// SIMATIC S7-200 project (STEP 7-Micro/WIN), CPU 226 CN REL 02.01

ORGANIZATION_BLOCK MAIN:OB1
TITLE=POU Comment
BEGIN
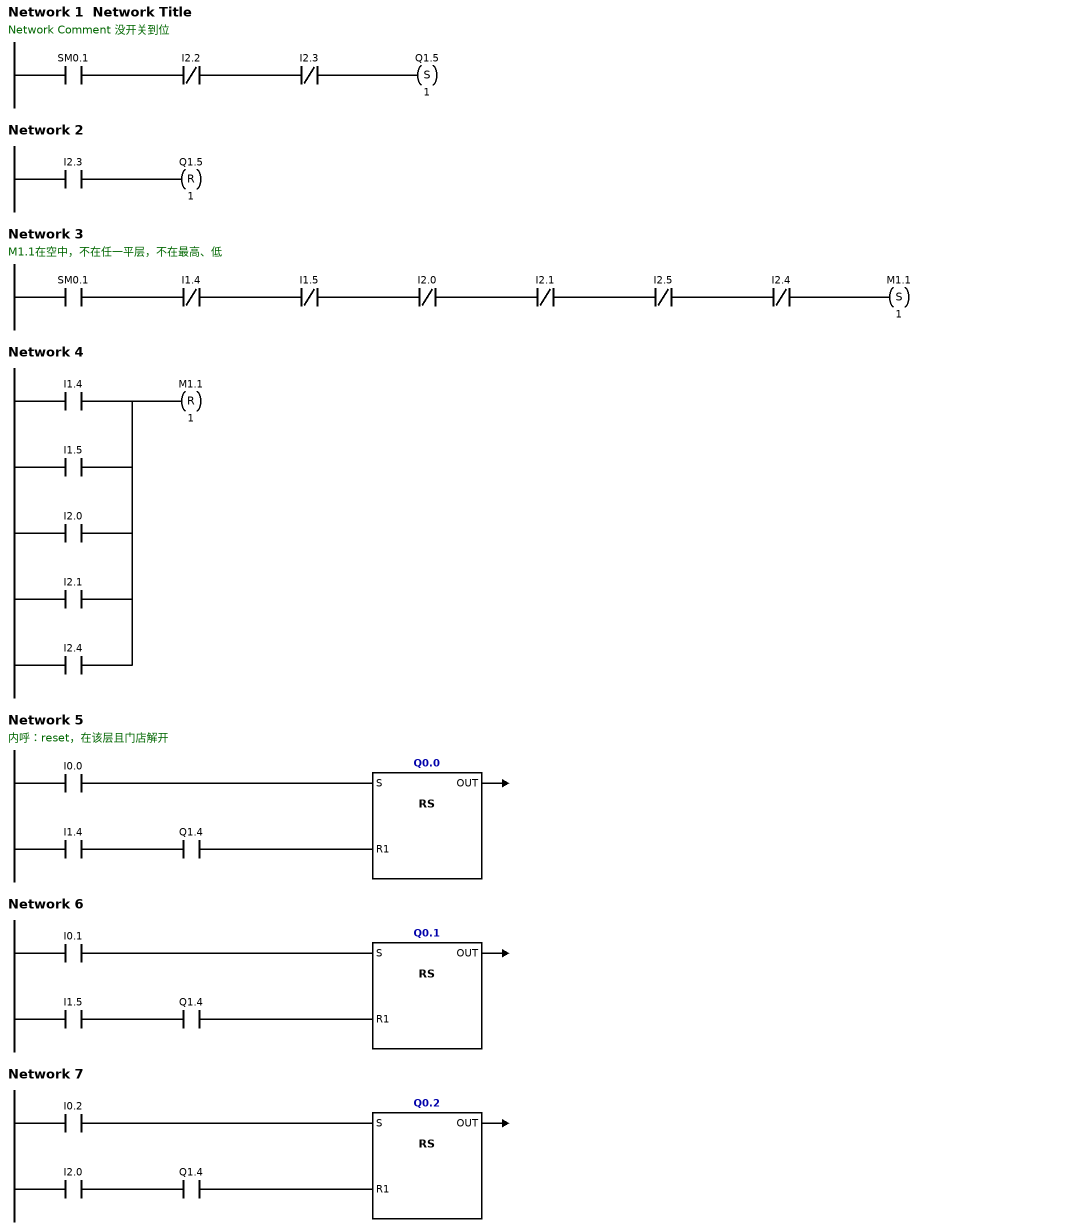
Network 1 // Network Title
// Network Comment 没开关到位
LD     SM0.1
AN     I2.2
AN     I2.3
S      Q1.5, 1
Network 2
LD     I2.3
R      Q1.5, 1
Network 3
// M1.1在空中，不在任一平层，不在最高、低
LD     SM0.1
AN     I1.4
AN     I1.5
AN     I2.0
AN     I2.1
AN     I2.5
AN     I2.4
S      M1.1, 1
Network 4
LD     I1.4
O      I1.5
O      I2.0
O      I2.1
O      I2.4
R      M1.1, 1
Network 5
// 内呼：reset，在该层且门店解开
LD     I0.0
LD     I1.4
A      Q1.4
NOT
LPS
A      Q0.0
=      Q0.0
LPP
ALD
O      Q0.0
=      Q0.0
Network 6
LD     I0.1
LD     I1.5
A      Q1.4
NOT
LPS
A      Q0.1
=      Q0.1
LPP
ALD
O      Q0.1
=      Q0.1
Network 7
LD     I0.2
LD     I2.0
A      Q1.4
NOT
LPS
A      Q0.2
=      Q0.2
LPP
ALD
O      Q0.2
=      Q0.2
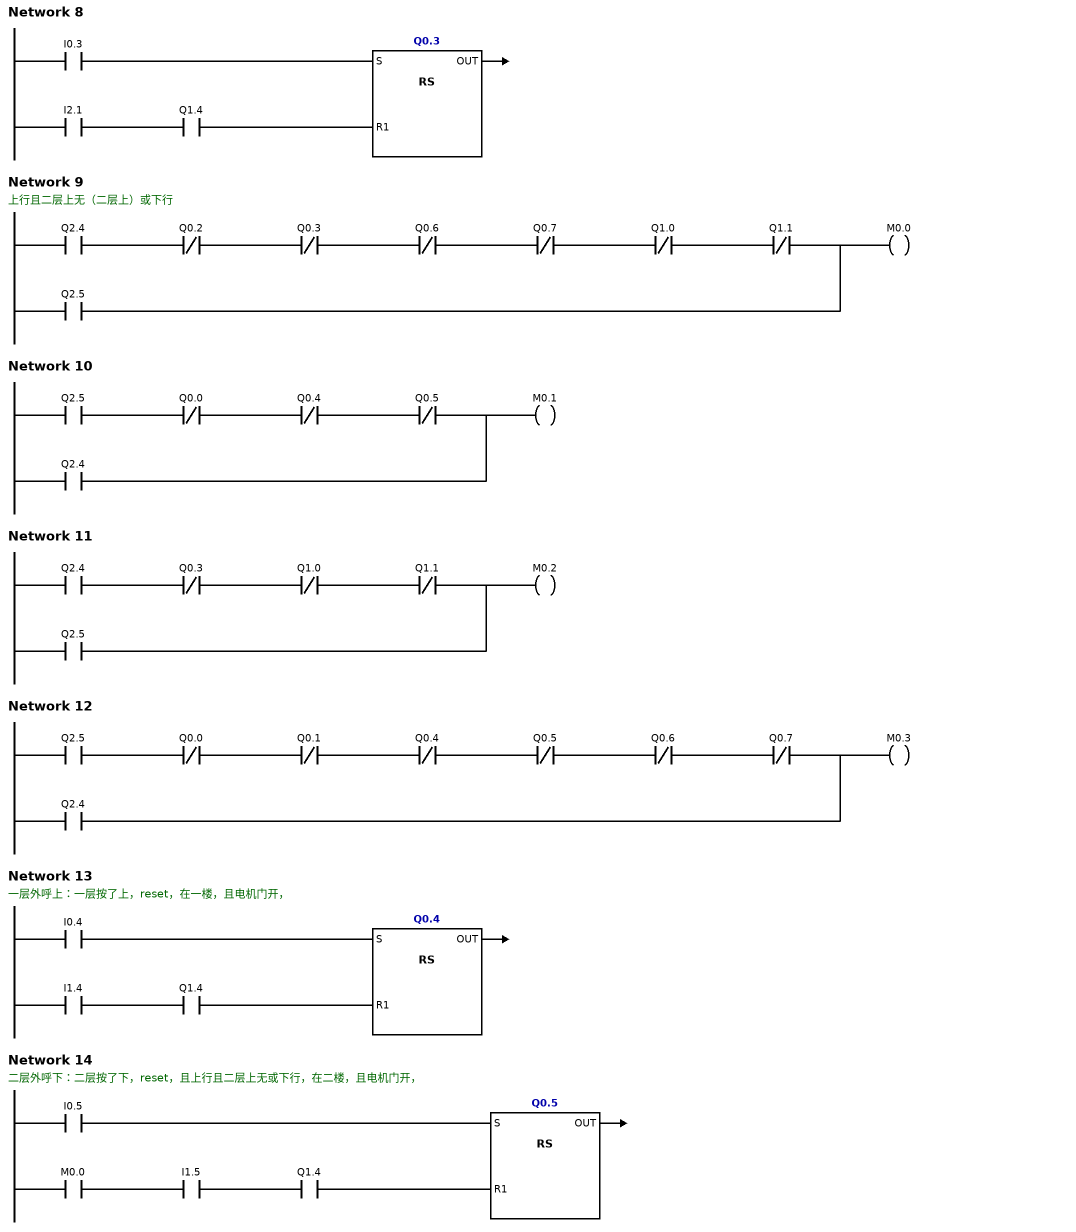
Network 8
LD     I0.3
LD     I2.1
A      Q1.4
NOT
LPS
A      Q0.3
=      Q0.3
LPP
ALD
O      Q0.3
=      Q0.3
Network 9
// 上行且二层上无（二层上）或下行
LD     Q2.4
AN     Q0.2
AN     Q0.3
AN     Q0.6
AN     Q0.7
AN     Q1.0
AN     Q1.1
O      Q2.5
=      M0.0
Network 10
LD     Q2.5
AN     Q0.0
AN     Q0.4
AN     Q0.5
O      Q2.4
=      M0.1
Network 11
LD     Q2.4
AN     Q0.3
AN     Q1.0
AN     Q1.1
O      Q2.5
=      M0.2
Network 12
LD     Q2.5
AN     Q0.0
AN     Q0.1
AN     Q0.4
AN     Q0.5
AN     Q0.6
AN     Q0.7
O      Q2.4
=      M0.3
Network 13
// 一层外呼上：一层按了上，reset，在一楼，且电机门开，
LD     I0.4
LD     I1.4
A      Q1.4
NOT
LPS
A      Q0.4
=      Q0.4
LPP
ALD
O      Q0.4
=      Q0.4
Network 14
// 二层外呼下：二层按了下，reset，且上行且二层上无或下行，在二楼，且电机门开，
LD     I0.5
LD     M0.0
A      I1.5
A      Q1.4
NOT
LPS
A      Q0.5
=      Q0.5
LPP
ALD
O      Q0.5
=      Q0.5
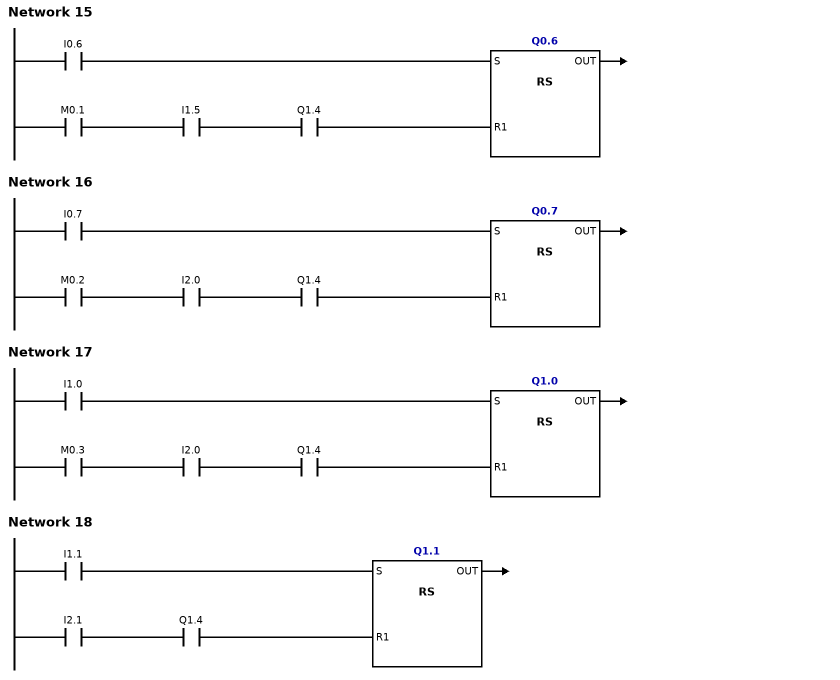
Network 15
LD     I0.6
LD     M0.1
A      I1.5
A      Q1.4
NOT
LPS
A      Q0.6
=      Q0.6
LPP
ALD
O      Q0.6
=      Q0.6
Network 16
LD     I0.7
LD     M0.2
A      I2.0
A      Q1.4
NOT
LPS
A      Q0.7
=      Q0.7
LPP
ALD
O      Q0.7
=      Q0.7
Network 17
LD     I1.0
LD     M0.3
A      I2.0
A      Q1.4
NOT
LPS
A      Q1.0
=      Q1.0
LPP
ALD
O      Q1.0
=      Q1.0
Network 18
LD     I1.1
LD     I2.1
A      Q1.4
NOT
LPS
A      Q1.1
=      Q1.1
LPP
ALD
O      Q1.1
=      Q1.1
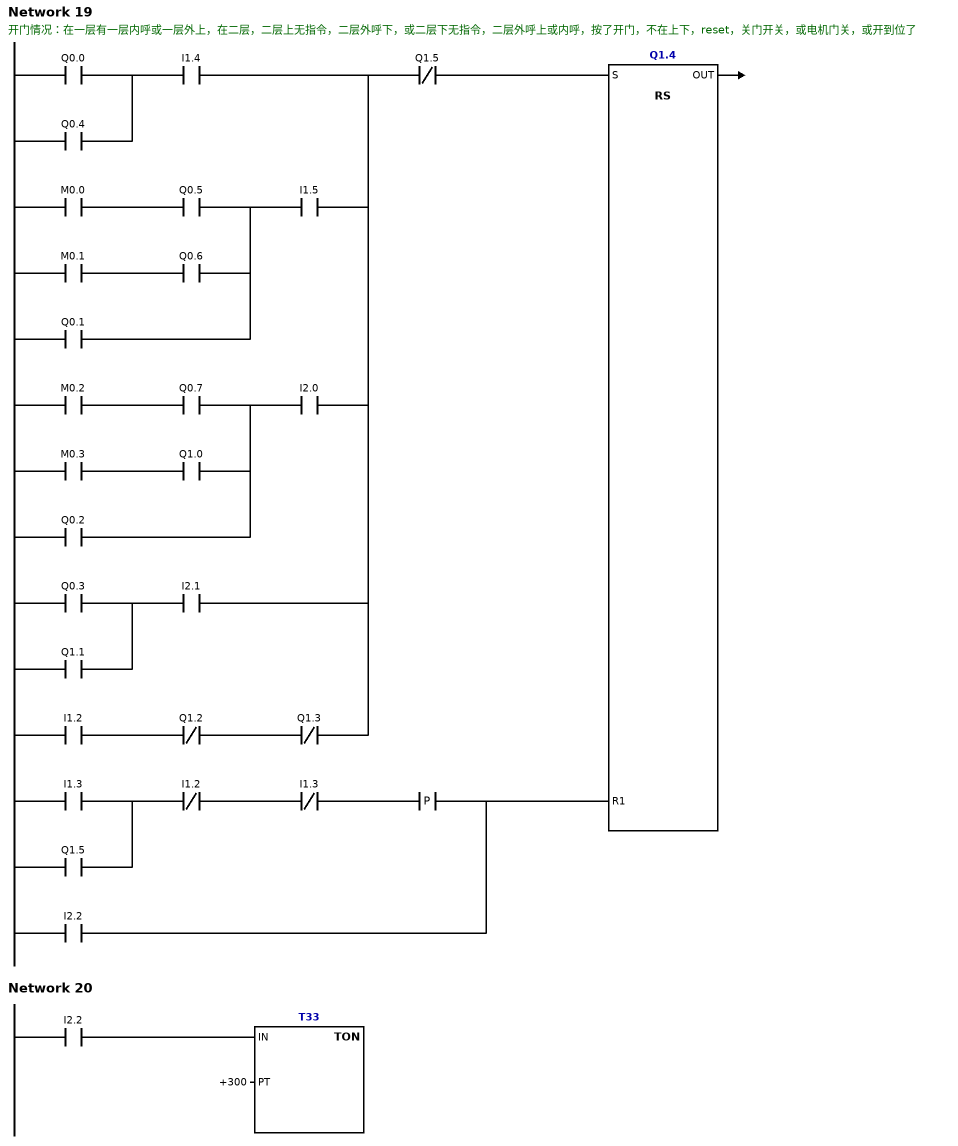
Network 19
// 开门情况：在一层有一层内呼或一层外上，在二层，二层上无指令，二层外呼下，或二层下无指令，二层外呼上或内呼，按了开门，不在上下，reset，关门开关，或电机门关，或开到位了
LD     Q0.0
O      Q0.4
A      I1.4
LD     M0.0
A      Q0.5
LD     M0.1
A      Q0.6
OLD
O      Q0.1
A      I1.5
OLD
LD     M0.2
A      Q0.7
LD     M0.3
A      Q1.0
OLD
O      Q0.2
A      I2.0
OLD
LD     Q0.3
O      Q1.1
A      I2.1
OLD
LD     I1.2
AN     Q1.2
AN     Q1.3
OLD
AN     Q1.5
LD     I1.3
O      Q1.5
AN     I1.2
AN     I1.3
EU
O      I2.2
NOT
LPS
A      Q1.4
=      Q1.4
LPP
ALD
O      Q1.4
=      Q1.4
Network 20
LD     I2.2
TON    T33, +300
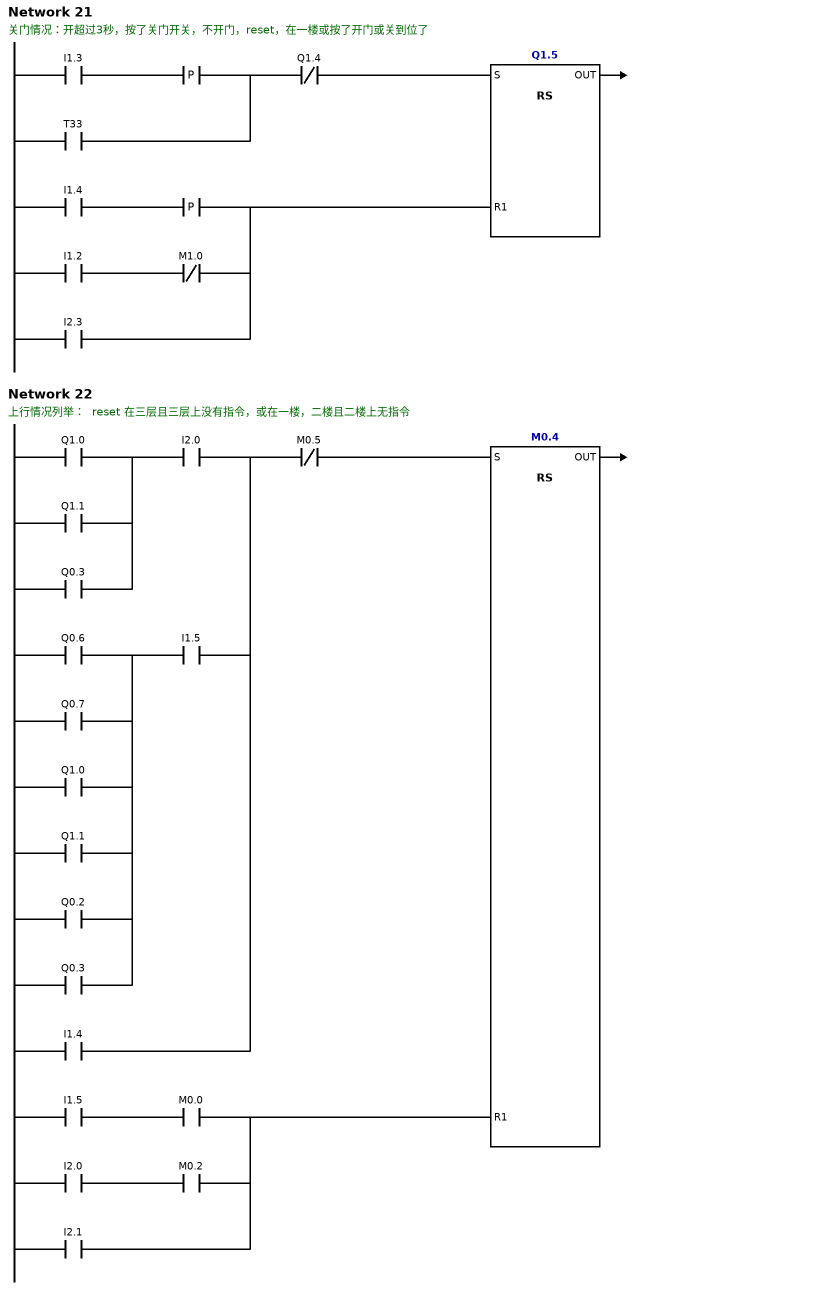
Network 21
// 关门情况：开超过3秒，按了关门开关，不开门，reset，在一楼或按了开门或关到位了
LD     I1.3
EU
O      T33
AN     Q1.4
LD     I1.4
EU
LD     I1.2
AN     M1.0
OLD
O      I2.3
NOT
LPS
A      Q1.5
=      Q1.5
LPP
ALD
O      Q1.5
=      Q1.5
Network 22
// 上行情况列举：  reset 在三层且三层上没有指令，或在一楼，二楼且二楼上无指令
LD     Q1.0
O      Q1.1
O      Q0.3
A      I2.0
LD     Q0.6
O      Q0.7
O      Q1.0
O      Q1.1
O      Q0.2
O      Q0.3
A      I1.5
OLD
O      I1.4
AN     M0.5
LD     I1.5
A      M0.0
LD     I2.0
A      M0.2
OLD
O      I2.1
NOT
LPS
A      M0.4
=      M0.4
LPP
ALD
O      M0.4
=      M0.4
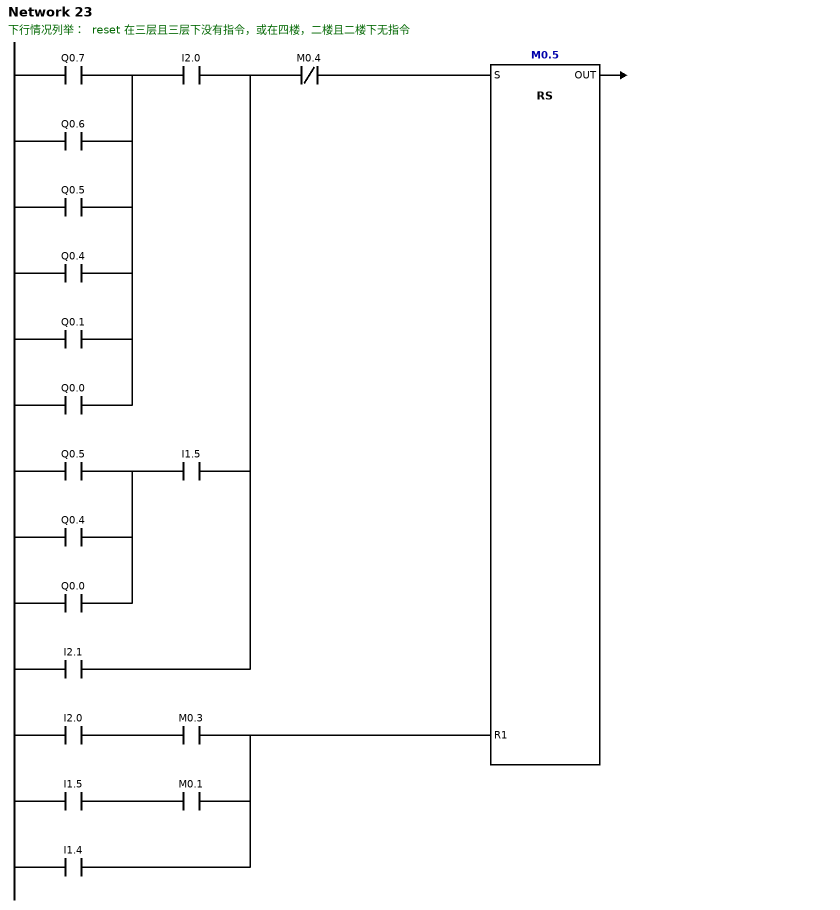
Network 23
// 下行情况列举：  reset 在三层且三层下没有指令，或在四楼，二楼且二楼下无指令
LD     Q0.7
O      Q0.6
O      Q0.5
O      Q0.4
O      Q0.1
O      Q0.0
A      I2.0
LD     Q0.5
O      Q0.4
O      Q0.0
A      I1.5
OLD
O      I2.1
AN     M0.4
LD     I2.0
A      M0.3
LD     I1.5
A      M0.1
OLD
O      I1.4
NOT
LPS
A      M0.5
=      M0.5
LPP
ALD
O      M0.5
=      M0.5
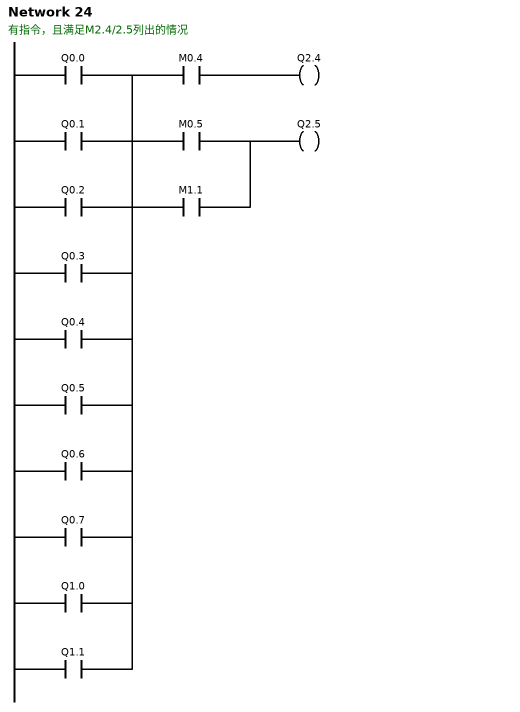
Network 24
// 有指令，且满足M2.4/2.5列出的情况
LD     Q0.0
O      Q0.1
O      Q0.2
O      Q0.3
O      Q0.4
O      Q0.5
O      Q0.6
O      Q0.7
O      Q1.0
O      Q1.1
LPS
A      M0.4
=      Q2.4
LPP
LD     M0.5
O      M1.1
ALD
=      Q2.5
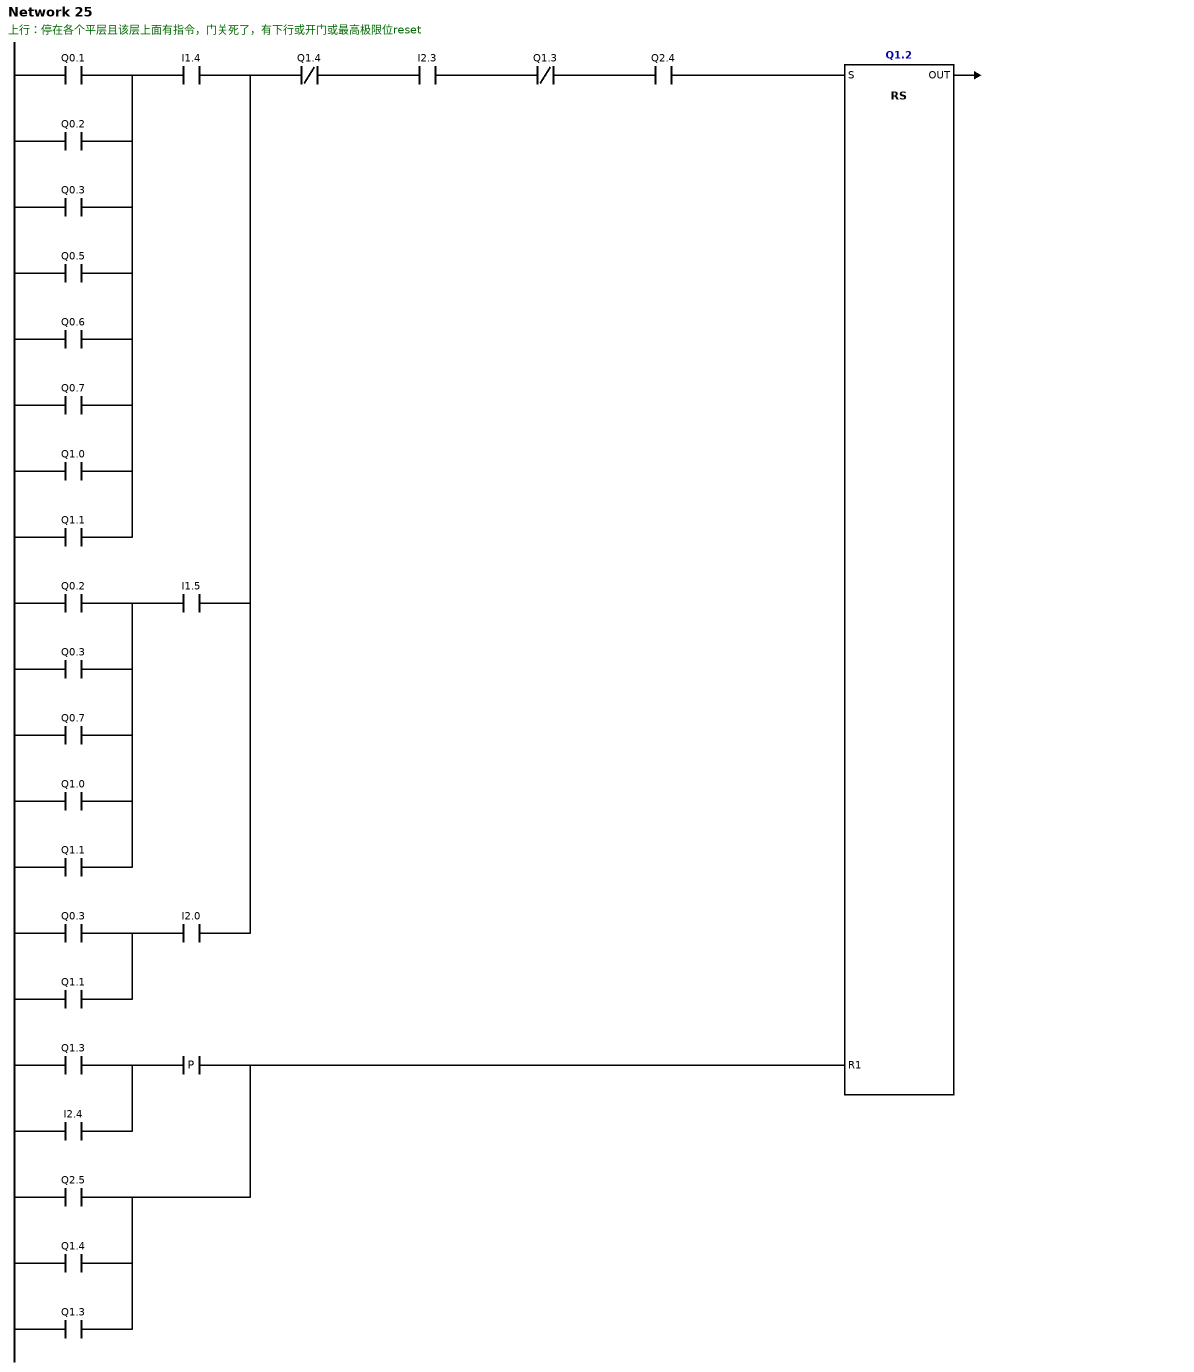
Network 25
// 上行：停在各个平层且该层上面有指令，门关死了，有下行或开门或最高极限位reset
LD     Q0.1
O      Q0.2
O      Q0.3
O      Q0.5
O      Q0.6
O      Q0.7
O      Q1.0
O      Q1.1
A      I1.4
LD     Q0.2
O      Q0.3
O      Q0.7
O      Q1.0
O      Q1.1
A      I1.5
OLD
LD     Q0.3
O      Q1.1
A      I2.0
OLD
AN     Q1.4
A      I2.3
AN     Q1.3
A      Q2.4
LD     Q1.3
O      I2.4
EU
LD     Q2.5
O      Q1.4
O      Q1.3
OLD
NOT
LPS
A      Q1.2
=      Q1.2
LPP
ALD
O      Q1.2
=      Q1.2
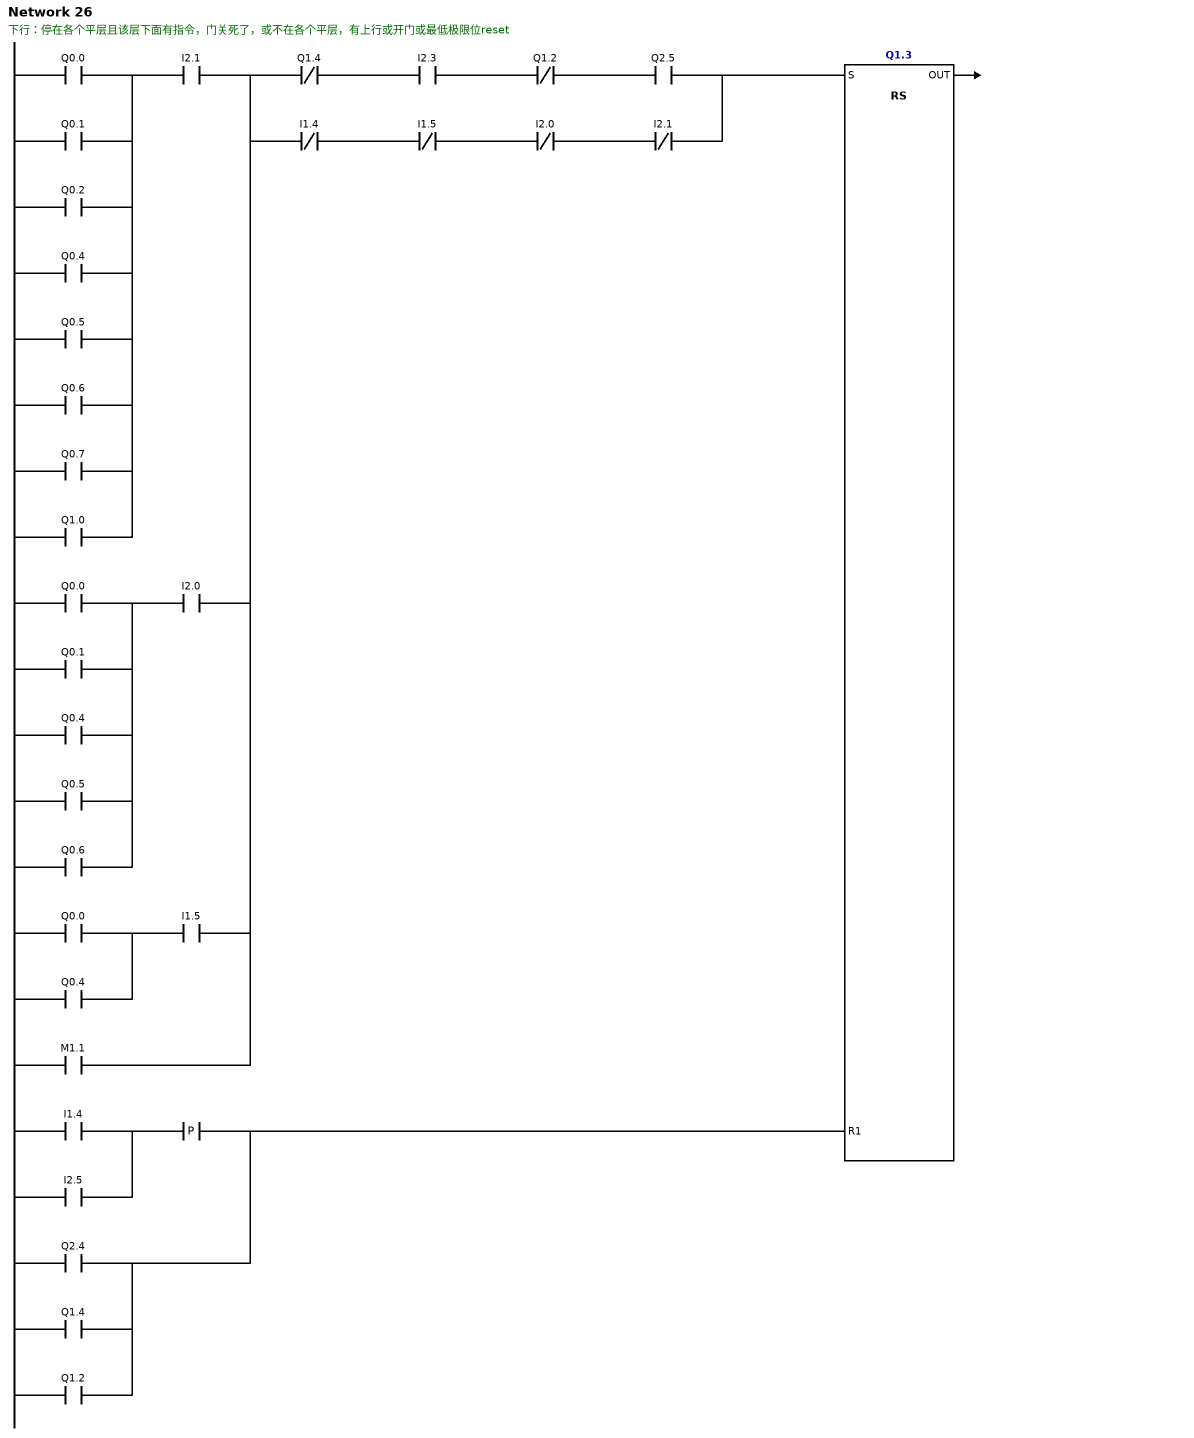
Network 26
// 下行：停在各个平层且该层下面有指令，门关死了，或不在各个平层，有上行或开门或最低极限位reset
LD     Q0.0
O      Q0.1
O      Q0.2
O      Q0.4
O      Q0.5
O      Q0.6
O      Q0.7
O      Q1.0
A      I2.1
LD     Q0.0
O      Q0.1
O      Q0.4
O      Q0.5
O      Q0.6
A      I2.0
OLD
LD     Q0.0
O      Q0.4
A      I1.5
OLD
O      M1.1
LDN    Q1.4
A      I2.3
AN     Q1.2
A      Q2.5
LDN    I1.4
AN     I1.5
AN     I2.0
AN     I2.1
OLD
ALD
LD     I1.4
O      I2.5
EU
LD     Q2.4
O      Q1.4
O      Q1.2
OLD
NOT
LPS
A      Q1.3
=      Q1.3
LPP
ALD
O      Q1.3
=      Q1.3
END_ORGANIZATION_BLOCK
